Universal Robots PolyScope program: sequential_p3.urp

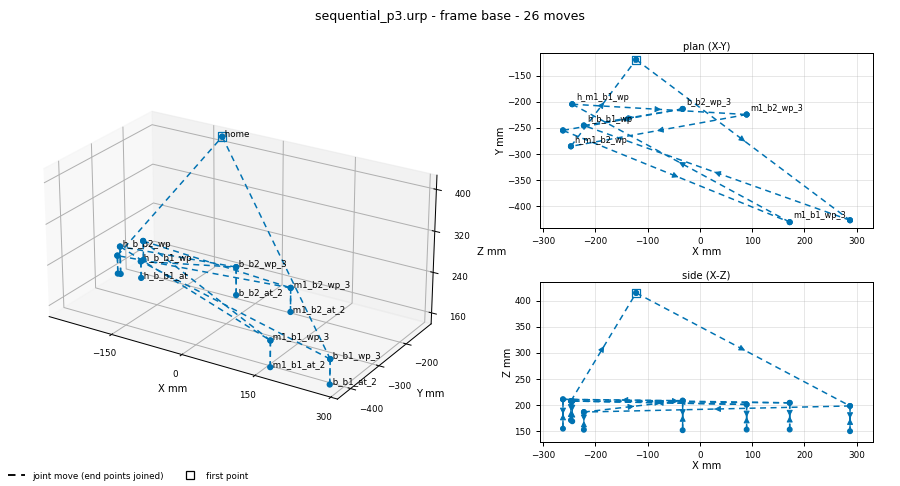
[picture p0: tool path of sequential_p3.urp in frame base, 26 of 26 moves have a stored position in this frame; points joined in program order, loops and branches not executed]
Program sequential_p3 (installation=default directory=/programs/usbdisk/ITER createdIn=5.3.1.64192 lastSavedIn=5.3.1.64192 robotSerialNumber=20195300365)
Calibrated DH parameters: a=[-0.000093, -0.190649, -0.212673, 0.000091, -0.000205, 0]; d=[0.151591, 44.061648, -42.488068, -1.442789, 0.085322, 0.091911]; alpha=[1.570082, -0.003447, 0.007513, 1.572293, -1.571904, 0]; deltaTheta=[0, -0.672656, 0.728185, -0.055522, 0.000005, 0]
Robot Program (runOnlyOnce=false)
  URCap Gripper Activate (Robotiq_Grippers, Robotiq Inc.) dataModel(ResetAndActivateKey=false)
  URCap Gripper (Robotiq_Grippers, Robotiq Inc.) dataModel(position=50.0, force=100.0, speed=100.0, positionInDouble=50.0, forceInDouble=100.0, speedInDouble=100.0, slaveIds=[9], blocking=true)
  MoveJ speed 60 deg/s, acceleration 80 deg/s^2 (useActiveTCP=true) feature=Base
    Waypoint home: TCP in base x=-122.15 y=-119.32 z=414.454 mm, rx=2.2563 ry=2.1459 rz=-0.0481 rad; joints [-85.681, -56.776, -79.802, -131.025, 89.944, -262.833] deg
  Folder Base
    MoveJ speed 60 deg/s, acceleration 80 deg/s^2 (useActiveTCP=true) feature=Base
      Waypoint b_b1_wp_3: TCP in base x=287.27 y=-426.687 z=198.703 mm, rx=2.2572 ry=2.1295 rz=-0.0633 rad; joints [-40.865, -143.306, -39.499, -85.215, 87.731, -217.488] deg
      Waypoint b_b1_at_2: TCP in base x=287.269 y=-426.683 z=150.489 mm, rx=2.2571 ry=2.1295 rz=-0.0633 rad; joints [-40.886, -145.62, -48.126, -74.275, 87.723, -217.437] deg
      URCap Gripper (Robotiq_Grippers, Robotiq Inc.) dataModel(position=100.0, force=100.0, speed=100.0, positionInDouble=100.0, forceInDouble=100.0, speedInDouble=100.0, slaveIds=[9], blocking=true)
      Waypoint b_b1_wp_4: TCP in base x=287.27 y=-426.687 z=198.703 mm, rx=2.2572 ry=2.1295 rz=-0.0633 rad; joints [-40.865, -143.306, -39.499, -85.215, 87.731, -217.488] deg
      Waypoint h_b_b1_wp: TCP in base x=-222.187 y=-245.349 z=187.06 mm, rx=-3.1315 ry=0.0204 rz=0.0123 rad; joints [-108.957, -99.116, -113.081, -58.146, 89.665, -197.782] deg
      Waypoint h_b_b1_at: TCP in base x=-222.188 y=-245.348 z=153.24 mm, rx=-3.1314 ry=0.0204 rz=0.0122 rad; joints [-108.969, -104.391, -117.643, -48.312, 89.612, -197.745] deg
      URCap Gripper (Robotiq_Grippers, Robotiq Inc.) dataModel(position=50.0, force=100.0, speed=100.0, positionInDouble=50.0, forceInDouble=100.0, speedInDouble=100.0, slaveIds=[9], blocking=true)
      Waypoint h_b_b1_wp: TCP in base x=-222.187 y=-245.349 z=187.06 mm, rx=-3.1315 ry=0.0204 rz=0.0123 rad; joints [-108.957, -99.116, -113.081, -58.146, 89.665, -197.782] deg
    MoveJ speed 60 deg/s, acceleration 80 deg/s^2 (useActiveTCP=true) feature=Base
      Waypoint b_b2_wp_3: TCP in base x=-33.1 y=-213.495 z=208.789 mm, rx=2.2331 ry=2.1669 rz=-0.0323 rad; joints [-61.64, -60.837, -137.744, -69.392, 89.733, -239.518] deg
      Waypoint b_b2_at_2: TCP in base x=-33.102 y=-213.489 z=152.337 mm, rx=2.2331 ry=2.167 rz=-0.0323 rad; joints [-61.683, -72.125, -150.112, -45.739, 89.609, -239.421] deg
      URCap Gripper (Robotiq_Grippers, Robotiq Inc.) dataModel(position=100.0, force=100.0, speed=100.0, positionInDouble=100.0, forceInDouble=100.0, speedInDouble=100.0, slaveIds=[9], blocking=true)
      Waypoint b_b2_wp_4: TCP in base x=-33.1 y=-213.495 z=208.789 mm, rx=2.2331 ry=2.1669 rz=-0.0323 rad; joints [-61.64, -60.837, -137.744, -69.392, 89.733, -239.518] deg
      Waypoint h_b_b2_wp: TCP in base x=-262.196 y=-254.726 z=211.351 mm, rx=-3.0605 ry=0.0443 rz=-0.0223 rad; joints [-114.749, -105.359, -96.042, -73.109, 89.199, -202.734] deg
      Waypoint h_b_b2_at: TCP in base x=-262.208 y=-254.718 z=155.33 mm, rx=-3.0605 ry=0.0443 rz=-0.0223 rad; joints [-114.774, -111.736, -104.192, -58.581, 89.146, -202.674] deg
      URCap Gripper (Robotiq_Grippers, Robotiq Inc.) dataModel(position=50.0, force=100.0, speed=100.0, positionInDouble=50.0, forceInDouble=100.0, speedInDouble=100.0, slaveIds=[9], blocking=true)
      Waypoint h_b_b2_wp: TCP in base x=-262.196 y=-254.726 z=211.351 mm, rx=-3.0605 ry=0.0443 rz=-0.0223 rad; joints [-114.749, -105.359, -96.042, -73.109, 89.199, -202.734] deg
  Folder Mid_1
    MoveJ speed 60 deg/s, acceleration 80 deg/s^2 (useActiveTCP=true) feature=Base
      Waypoint m1_b1_wp_3: TCP in base x=171.816 y=-430.356 z=204.684 mm, rx=2.26 ry=2.1667 rz=-0.0282 rad; joints [-51.724, -128.073, -65.156, -76.01, 89.303, -229.106] deg
      Waypoint m1_b1_at_2: TCP in base x=171.786 y=-430.365 z=153.694 mm, rx=2.2601 ry=2.1667 rz=-0.0282 rad; joints [-51.746, -132.202, -72.305, -64.735, 89.276, -229.058] deg
      URCap Gripper (Robotiq_Grippers, Robotiq Inc.) dataModel(position=100.0, force=100.0, speed=100.0, positionInDouble=100.0, forceInDouble=100.0, speedInDouble=100.0, slaveIds=[9], blocking=true)
      Waypoint m1_b1_wp_4: TCP in base x=171.816 y=-430.356 z=204.684 mm, rx=2.26 ry=2.1667 rz=-0.0282 rad; joints [-51.724, -128.073, -65.156, -76.01, 89.303, -229.106] deg
      Waypoint h_m1_b1_wp: TCP in base x=-244.449 y=-204.582 z=208.1 mm, rx=2.2684 ry=2.1196 rz=0.0229 rad; joints [-116.825, -93.932, -112.747, -63.308, 92.582, -292.535] deg
      Waypoint h_m1_b1_at: TCP in base x=-244.447 y=-204.577 z=169.457 mm, rx=2.2685 ry=2.1196 rz=0.0229 rad; joints [-116.841, -99.299, -118.834, -51.852, 92.525, -292.487] deg
      URCap Gripper (Robotiq_Grippers, Robotiq Inc.) dataModel(position=50.0, force=100.0, speed=100.0, positionInDouble=50.0, forceInDouble=100.0, speedInDouble=100.0, slaveIds=[9], blocking=true)
      Waypoint h_m1_b1_wp: TCP in base x=-244.449 y=-204.582 z=208.1 mm, rx=2.2684 ry=2.1196 rz=0.0229 rad; joints [-116.825, -93.932, -112.747, -63.308, 92.582, -292.535] deg
    MoveJ speed 60 deg/s, acceleration 80 deg/s^2 (useActiveTCP=true) feature=Base
      Waypoint m1_b2_wp_3: TCP in base x=89.366 y=-224.31 z=201.565 mm, rx=-2.2386 ry=-2.1806 rz=-0.0102 rad; joints [-36.103, -72.547, -132.567, -65.683, 90.9, -214.176] deg
      Waypoint m1_b2_at_2: TCP in base x=89.368 y=-224.313 z=153.584 mm, rx=-2.2387 ry=-2.1806 rz=-0.0101 rad; joints [-36.132, -81.828, -141.776, -47.193, 90.798, -214.098] deg
      URCap Gripper (Robotiq_Grippers, Robotiq Inc.) dataModel(position=100.0, force=100.0, speed=100.0, positionInDouble=100.0, forceInDouble=100.0, speedInDouble=100.0, slaveIds=[9], blocking=true)
      Waypoint m1_b2_wp_4: TCP in base x=89.366 y=-224.31 z=201.565 mm, rx=-2.2386 ry=-2.1806 rz=-0.0102 rad; joints [-36.103, -72.547, -132.567, -65.683, 90.9, -214.176] deg
      Waypoint h_m1_b2_wp: TCP in base x=-247.009 y=-285.144 z=208.116 mm, rx=2.2684 ry=2.1195 rz=0.0229 rad; joints [-111.389, -107.719, -95.772, -66.28, 92.556, -287.152] deg
      Waypoint h_m1_b2_at: TCP in base x=-246.994 y=-285.166 z=171.647 mm, rx=2.2684 ry=2.1196 rz=0.0229 rad; joints [-111.399, -111.783, -101.037, -56.949, 92.516, -287.113] deg
      URCap Gripper (Robotiq_Grippers, Robotiq Inc.) dataModel(position=50.0, force=100.0, speed=100.0, positionInDouble=50.0, forceInDouble=100.0, speedInDouble=100.0, slaveIds=[9], blocking=true)
      Waypoint h_m1_b2_wp: TCP in base x=-247.009 y=-285.144 z=208.116 mm, rx=2.2684 ry=2.1195 rz=0.0229 rad; joints [-111.389, -107.719, -95.772, -66.28, 92.556, -287.152] deg
  MoveJ speed 60 deg/s, acceleration 80 deg/s^2 (useActiveTCP=true) feature=Base
    Waypoint home: TCP in base x=-122.15 y=-119.32 z=414.454 mm, rx=2.2563 ry=2.1459 rz=-0.0481 rad; joints [-85.681, -56.776, -79.802, -131.025, 89.944, -262.833] deg
